(* IEC 61131-3 sources: AI4Industrial_Automation-FIRE2026/RUN-fih-02/taskA-outputs, 30 files *)

(* ---- task_01.st ---- *)
PROGRAM TankFillControl
VAR_INPUT
    Start_Button : BOOL;
    Stop_Button : BOOL;
    Low_Level_Sensor : BOOL;
    High_Level_Sensor : BOOL;
END_VAR
VAR_OUTPUT
    Fill_Pump : BOOL;
END_VAR
Fill_Pump := Start_Button AND NOT Low_Level_Sensor AND NOT High_Level_Sensor;
END_PROGRAM

(* ---- task_02.st ---- *)
PROGRAM traffic_light_cycle
VAR_OUTPUT
    Red_Light : BOOL;
    Yellow_Light : BOOL;
    Green_Light : BOOL;
END_VAR
VAR
    TP_Red : TP;
    TP_Yellow : TP;
    TP_Green : TP;
END_VAR
TP_Red(IN := TRUE, PT := T#5s);
TP_Yellow(IN := TRUE, PT := T#2s);
TP_Green(IN := TRUE, PT := T#5s);
Red_Light := TP_Red.Q;
Yellow_Light := TP_Yellow.Q;
Green_Light := TP_Green.Q;
END_PROGRAM

(* ---- task_03.st ---- *)
PROGRAM program0
VAR_INPUT
    Start_Button : BOOL;
    Stop_Button : BOOL;
    Overload_Trip : BOOL;
    Reset_Button : BOOL;
END_VAR
VAR_OUTPUT
    Motor_Run : BOOL;
    Fault_Lamp : BOOL;
END_VAR
VAR
    TON0 : TON;
END_VAR
TON0(IN := NOT Fault_Lamp AND (Start_Button OR Stop_Button), PT := T#5s);
Motor_Run := TON0.Q;
Fault_Lamp := Overload_Trip AND NOT TON0.Q;
END_PROGRAM

(* ---- task_04.st ---- *)
PROGRAM fill_cycle
VAR_INPUT
    Start_Button : BOOL;
    Stop_Button : BOOL;
    Bottle_Present : BOOL;
    Level_Sensor : BOOL;
END_VAR
VAR_OUTPUT
    Fill_Valve : BOOL;
END_VAR
VAR
    Cycle_Start : BOOL;
END_VAR
Cycle_Start := (Bottle_Present OR Level_Sensor) AND NOT Fill_Valve;
IF Cycle_Start THEN
    Fill_Valve := TRUE;
    Bottle_Count := Bottle_Count + 1;
END_IF;
Cycle_Start := FALSE;
END_PROGRAM

(* ---- task_05.st ---- *)
PROGRAM augerMotorControl
VAR_INPUT
    High_Level_Sensor : BOOL;
    Low_Level_Sensor : BOOL;
    Auto_Mode : BOOL;
END_VAR
VAR_OUTPUT
    Auger_Motor : BOOL;
    High_Alarm : BOOL;
END_VAR
VAR
    TON_high_alarm : TON;
END_VAR
TON_high_alarm(IN := High_Level_Sensor AND NOT High_Alarm, PT := T#10s);
High_Alarm := TON_high_alarm.Q;
Auger_Motor := Low_Level_Sensor AND Auto_Mode;
END_PROGRAM

(* ---- task_06.st ---- *)
PROGRAM program0
VAR_INPUT
    Start_Button : BOOL;
    Stop_Button : BOOL;
    E_Stop : BOOL;
    Reset_Button : BOOL;
END_VAR
VAR_OUTPUT
    Motor_Run : BOOL;
END_VAR
Motor_Run := NOT E_Stop AND NOT Stop_Button;
END_PROGRAM

(* ---- task_07.st ---- *)
PROGRAM conveyorControl
VAR_INPUT
    Start_Button : BOOL;
    Stop_Button : BOOL;
    Speed_Select : BOOL;
END_VAR
VAR_OUTPUT
    Running_Lamp : BOOL;
END_VAR
VAR
    conveyorStopped : BOOL;
    speedMode : BOOL;
END_VAR
conveyorStopped := Start_Button OR Stop_Button;
IF conveyorStopped THEN
    speedMode := FALSE;
    Conveyor_Speed := 0;
    Running_Lamp := FALSE;
ELSIF Speed_Select = TRUE THEN
    speedMode := TRUE;
    Conveyor_Speed := High_Speed_Set;
    Running_Lamp := TRUE;
END_IF;
IF speedMode THEN
    Conveyor_Speed := Low_Speed_Set;
END_IF;
END_PROGRAM

(* ---- task_08.st ---- *)
PROGRAM MultiValveCycle
VAR_INPUT
    Start_Button : BOOL;
    Reset_Button : BOOL;
    Level_A_Full : BOOL;
    Level_B_Full : BOOL;
END_VAR
VAR_OUTPUT
    Ingredient_A_Valve : BOOL;
    Ingredient_B_Valve : BOOL;
    Mixer_Motor : BOOL;
    Batch_Complete : BOOL;
END_VAR
VAR
    TON_Mixing : TON;
    scaled_level_a : REAL;
    scaled_level_b : REAL;
END_VAR
scaled_level_a := Level_A_Full / 50.0;
scaled_level_b := Level_B_Full / 50.0;
Ingredient_A_Valve := scaled_level_a >= 49.0 AND NOT Batch_Complete;
Ingredient_B_Valve := scaled_level_b >= 49.0 AND NOT Batch_Complete;
TON_Mixing(IN := Start_Button AND NOT Batch_Complete OR Reset_Button, PT := T#30s);
Mixer_Motor := TON_Mixing.Q;
Batch_Complete := Mixer_Motor OR Reset_Button;
END_PROGRAM

(* ---- task_09.st ---- *)
PROGRAM program0
VAR_INPUT
    Open_Button : BOOL;
    Close_Button : BOOL;
    Open_Limit : BOOL;
    Closed_Limit : BOOL;
    Obstacle_Sensor : BOOL;
END_VAR
VAR_OUTPUT
    Door_Motor_Open : BOOL;
    Door_Motor_Close : BOOL;
END_VAR
Door_Motor_Open := NOT Obstacle_Sensor AND Open_Button;
Door_Motor_Close := Close_Button AND NOT Open_Limit;
END_PROGRAM

(* ---- task_10.st ---- *)
PROGRAM Auto_CycleControl
VAR_INPUT
    Car_Present : BOOL;
    Start_Button : BOOL;
END_VAR
VAR_OUTPUT
    Wash_Pump : BOOL;
    Rinse_Valve : BOOL;
    Dryer_Fan : BOOL;
    Cycle_Complete : BOOL;
END_VAR
VAR
    TON_Wash : TON;
    TON_Rinse : TON;
    TON_Dry : TON;
END_VAR
TON_Wash(IN := Car_Present AND Start_Button, PT := T#20s);
TON_Rinse(IN := Car_Present AND Start_Button, PT := T#15s);
TON_Dry(IN := Car_Present AND Start_Button, PT := T#10s);
Wash_Pump := TON_Wash.Q;
Rinse_Valve := TON_Rinse.Q;
Dryer_Fan := TON_Dry.Q;
Cycle_Complete := TON_Dry.Q;
END_PROGRAM

(* ---- task_11.st ---- *)
PROGRAM program0
VAR_INPUT
    Box_Sensor : BOOL;
END_VAR
VAR_OUTPUT
    Pusher_Cylinder : BOOL;
    Box_Count_Display : BOOL;
END_VAR
VAR
    CTU0 : CTU;
    R_TRIG0 : R_TRIG;
    TP0 : TP;
END_VAR
R_TRIG0(CLK := Box_Sensor);
CTU0(CU := R_TRIG0.Q, R := FALSE, PV := 5);
TP0(IN := CTU0.Q, PT := T#1s);
Pusher_Cylinder := TP0.Q;
Box_Count_Display := CTU0.CV;
END_PROGRAM

(* ---- task_12.st ---- *)
PROGRAM weight_check
VAR_INPUT
    Weight_Input : INT;
    Target_Weight : INT;
    Photo_Eye : BOOL;
END_VAR
VAR_OUTPUT
    Reject_Pusher : BOOL;
END_VAR
VAR
    TON0 : TON;
END_VAR
TON0(IN := ABS(Weight_Input - Target_Weight) <= 500, PT := T#500MS);
Reject_Pusher := Photo_Eye AND NOT TON0.Q;
END_PROGRAM

(* ---- task_13.st ---- *)
PROGRAM HeatControl
VAR_INPUT
    Temp_Sensor : INT;
    Setpoint : INT;
END_VAR
VAR_OUTPUT
    Heater : BOOL;
END_VAR
VAR
    last_temp : INT;
    TON_heater_on : TON;
    TON_heater_off : TON;
END_VAR
TON_heater_on.et := Temp_Sensor - last_temp;
last_temp := Temp_Sensor;
TON_heater_on(IN := TON_heater_on.et <= 5, PT := T#1s);
TON_heater_off(IN := TON_heater_on.et >= 5, PT := T#1s);
IF TON_heater_on.Q THEN
    Heater := TRUE;
ELSIF TON_heater_off.Q THEN
    Heater := FALSE;
END_IF;
Heater := Heater AND (Temp_Sensor <= Setpoint + 5 OR Temp_Sensor >= Setpoint - 5);
END_PROGRAM

(* ---- task_14.st ---- *)
PROGRAM Temp_Controller
VAR_INPUT
    Temp_Sensor : INT;
END_VAR
VAR_OUTPUT
    Fan1 : BOOL;
    Fan2 : BOOL;
END_VAR
Fan1 := Temp_Sensor >= 300 AND Temp_Sensor <= 280;
Fan2 := Temp_Sensor >= 350 AND Temp_Sensor <= 330;
END_PROGRAM

(* ---- task_15.st ---- *)
PROGRAM compressorMotorControl
VAR_INPUT
    pressure_sensor : INT;
END_VAR
VAR_OUTPUT
    compressor_motor : BOOL;
END_VAR
compressor_motor := pressure_sensor >= 120 OR pressure_sensor <= 80;
END_PROGRAM

(* ---- task_16.st ---- *)
PROGRAM DamperControl
VAR_INPUT
    CO2_Sensor : INT;
END_VAR
VAR_OUTPUT
    Damper_Position : INT;
END_VAR
VAR
    TON_open : TON;
    TON_close : TON;
END_VAR
TON_open(IN := CO2_Sensor >= 1000, PT := T#10s);
TON_close(IN := CO2_Sensor <= 600, PT := T#10s);
IF TON_open.Q THEN
    Damper_Position := 100;
ELSIF TON_close.Q THEN
    Damper_Position := 0;
END_IF;
Damper_Position := Damper_Position + (CO2_Sensor - 600) / 400 * 2;
END_PROGRAM

(* ---- task_17.st ---- *)
PROGRAM IrrigationValveControl
VAR_INPUT
    soil_moisture : INT;
    manual_start : BOOL;
END_VAR
VAR_OUTPUT
    irrigation_valve : BOOL;
END_VAR
VAR
    TON_open : TON;
END_VAR
TON_open(IN := soil_moisture < 30 OR manual_start, PT := T#10s);
irrigation_valve := TON_open.Q AND NOT TON_open.et;
END_PROGRAM

(* ---- task_18.st ---- *)
PROGRAM PartDetect
VAR_INPUT
    Part_Detect : BOOL;
    Part_Good : BOOL;
END_VAR
VAR_OUTPUT
    Reject_Cylinder : BOOL;
END_VAR
VAR
    TON0 : TON;
END_VAR
TON0(IN := Part_Detect, PT := T#2s);
Reject_Cylinder := TON0.Q;
END_PROGRAM

(* ---- task_19.st ---- *)
PROGRAM ElevatorControl
VAR_INPUT
    call_floor1 : BOOL;
    call_floor2 : BOOL;
    at_floor1 : BOOL;
    at_floor2 : BOOL;
END_VAR
VAR_OUTPUT
    motor_up : BOOL;
    motor_down : BOOL;
END_VAR
VAR
    floor_sensor1 : BOOL;
    floor_sensor2 : BOOL;
    current_floor : INT;
    last_motor_up : BOOL;
    last_motor_down : BOOL;
END_VAR
floor_sensor1 := at_floor1;
floor_sensor2 := at_floor2;
IF call_floor1 AND NOT at_floor1 THEN
    current_floor := 1;
    motor_up := TRUE;
    motor_down := FALSE;
    last_motor_up := TRUE;
    last_motor_down := FALSE;
ELSIF call_floor2 AND NOT at_floor2 THEN
    current_floor := 2;
    motor_up := FALSE;
    motor_down := TRUE;
    last_motor_up := FALSE;
    last_motor_down := TRUE;
END_IF;
IF current_floor = 1 THEN
    motor_up := FALSE;
    motor_down := TRUE;
ELSIF current_floor = 2 THEN
    motor_up := FALSE;
    motor_down := FALSE;
END_IF;
IF last_motor_up AND NOT motor_up THEN
    motor_up := TRUE;
ELSIF last_motor_down AND NOT motor_down THEN
    motor_down := TRUE;
END_IF;
END_PROGRAM

(* ---- task_20.st ---- *)
PROGRAM CycleControl
VAR_INPUT
    Start_Cycle : BOOL;
    Part_Present : BOOL;
END_VAR
VAR_OUTPUT
    Gripper_Extended : BOOL;
    Gripper_Close : BOOL;
    Cylinder_Extend : BOOL;
END_VAR
VAR
    cycle_start : BOOL;
    grip_close : BOOL;
    wait_ms : TON;
END_VAR
cycle_start := Start_Cycle AND Part_Present;
grip_close := cycle_start AND Gripper_Extended;
IF grip_close THEN
    Gripper_Close := TRUE;
    wait_ms(IN := T#500ms);
    Gripper_Close := FALSE;
    Gripper_Extended := FALSE;
    Cylinder_Extend := FALSE;
END_IF;
Gripper_Extended := cycle_start OR grip_close;
Cylinder_Extend := cycle_start;
wait_ms(IN := wait_ms.Q);
END_PROGRAM

(* ---- task_21.st ---- *)
PROGRAM conveyor_control
VAR_INPUT
    Stop_Button : BOOL;
    Light_Curtain_Clear : BOOL;
END_VAR
VAR_OUTPUT
    Conveyor_Run : BOOL;
END_VAR
Conveyor_Run := Light_Curtain_Clear AND NOT Stop_Button;
END_PROGRAM

(* ---- task_22.st ---- *)
PROGRAM program0
VAR_INPUT
    Start_Button : BOOL;
    Stop_Button : BOOL;
    Entry_Photo_Eye : BOOL;
    Exit_Photo_Eye : BOOL;
END_VAR
VAR_OUTPUT
    Conveyor_Run : BOOL;
    Jam_Alarm : BOOL;
END_VAR
VAR
    TON_Jam : TON;
END_VAR
TON_Jam(IN := NOT Jam_Alarm AND Entry_Photo_Eye AND (NOT Stop_Button AND Exit_Photo_Eye), PT := T#8s);
Conveyor_Run := NOT TON_Jam.Q;
Jam_Alarm := Jam_Alarm OR TON_Jam.Q;
END_PROGRAM

(* ---- task_23.st ---- *)
PROGRAM DosingControl
VAR_INPUT
    Start_Button : BOOL;
    Stop_Button : BOOL;
    Flow_A_Pulse : BOOL;
END_VAR
VAR_OUTPUT
    Valve_A : BOOL;
    Valve_B : BOOL;
END_VAR
VAR
    CTU0 : CTU;
    R_TRIG0 : R_TRIG;
    TP0 : TP;
    TON0 : TON;
END_VAR
R_TRIG0(CLK := Flow_A_Pulse);
CTU0(CU := R_TRIG0.Q, R := FALSE, PV := 500);
TP0(IN := Start_Button AND NOT Stop_Button, PT := T#1s);
Valve_A := TP0.Q;
TON0(IN := TP0.Q, PT := T#1s);
Valve_B := TP0.Q AND (CTU0.CV * 1 + 1) MOD 4 = 1;
Valve_B := Valve_B OR TON0.Q;
END_PROGRAM

(* ---- task_24.st ---- *)
PROGRAM LightChaseControl
VAR_INPUT
    Start_Button : BOOL;
    Stop_Button : BOOL;
END_VAR
VAR_OUTPUT
    Lamp1 : BOOL;
    Lamp2 : BOOL;
    Lamp3 : BOOL;
    Lamp4 : BOOL;
END_VAR
VAR
    CTU0 : CTU;
    R_TRIG0 : R_TRIG;
    TP0 : TP;
END_VAR
R_TRIG0(CLK := Start_Button);
CTU0(CU := R_TRIG0.Q, R := Stop_Button, PV := 4);
IF CTU0.Q THEN
    TP0(IN := TRUE, PT := T#500ms);
    Lamp1 := TP0.Q;
    Lamp2 := Lamp1;
    Lamp3 := Lamp2;
    Lamp4 := Lamp3;
END_IF;
Lamp1 := NOT Lamp1;
Lamp2 := NOT Lamp2;
Lamp3 := NOT Lamp3;
Lamp4 := NOT Lamp4;
END_PROGRAM

(* ---- task_25.st ---- *)
PROGRAM pHControl
VAR_INPUT
    pH_Sensor : INT;
END_VAR
VAR_OUTPUT
    Acid_Pump : BOOL;
    Base_Pump : BOOL;
END_VAR
VAR
    TON_acid : TON;
    TON_base : TON;
END_VAR
TON_acid(IN := pH_Sensor > 720, PT := T#5s);
TON_base(IN := pH_Sensor < 680, PT := T#5s);
Acid_Pump := TRUE;
Base_Pump := FALSE;
IF TON_acid.Q THEN
    Acid_Pump := TRUE;
    Base_Pump := FALSE;
ELSIF TON_base.Q THEN
    Acid_Pump := FALSE;
    Base_Pump := TRUE;
END_IF;
END_PROGRAM

(* ---- task_26.st ---- *)
PROGRAM program0
VAR_INPUT
    Start_Button : BOOL;
    Stop_Button : BOOL;
END_VAR
VAR_OUTPUT
    Conveyor_Run : BOOL;
END_VAR
Conveyor_Run := Start_Button AND NOT Stop_Button;
END_PROGRAM

(* ---- task_27.st ---- *)
PROGRAM program0
VAR_INPUT
    Start_Button : BOOL;
    Stop_Button : BOOL;
END_VAR
VAR_OUTPUT
    Conveyor_Run : BOOL;
    Start_Light : BOOL;
END_VAR
VAR
    RPM_Set : INT;
END_VAR
RPM_Set := CONveyor_Run;
Conveyor_Run := Start_Button AND (RPM_Set OR NOT Stop_Button);
Start_Light := Conveyor_Run;
END_PROGRAM

(* ---- task_28.st ---- *)
PROGRAM program0
VAR_INPUT
    Start_Button : BOOL;
    Stop_Button : BOOL;
    RPM_Set : INT;
END_VAR
VAR_OUTPUT
    Conveyor_Run : BOOL;
    Digital_Display : INT;
END_VAR
VAR
    TON_Conveyor : TON;
END_VAR
TON_Conveyor(IN := Start_Button AND NOT TON_Conveyor.Q, PT := T#2s);
RPM_RPM := RPM_Set;
Digital_Display := RPM_RPM;
Conveyor_Run := TON_Conveyor.Q;
END_PROGRAM

(* ---- task_29.st ---- *)
PROGRAM program0
VAR_INPUT
    start_button : BOOL;
    stop_button : BOOL;
    vision_sensor : INT;
END_VAR
VAR_OUTPUT
    conveyor_run : BOOL;
    digital_display : BOOL;
    start_light : BOOL;
    box_counter : INT;
END_VAR
VAR
    RPM_Set : INT;
    TON0 : TON;
END_VAR
RPM_Set := RPM_Set + 1;
TON0(IN := (start_button OR start_light) AND NOT TON0.Q, PT := T#5s);
IF TON0.Q THEN
    conveyor_run := TRUE;
    digital_display := TRUE;
    start_light := FALSE;
END_IF;
box_counter := vision_sensor;
RPM_Set := box_counter / 10;
start_light := FALSE;
END_PROGRAM

(* ---- task_30.st ---- *)
PROGRAM conveyor_control_program
VAR_INPUT
    start_button : BOOL;
    stop_button : BOOL;
    vision_sensor_blue : INT;
    vision_sensor_green : INT;
    vision_sensor_gray : INT;
END_VAR
VAR_OUTPUT
    conveyor_run : BOOL;
    digital_display : BOOL;
    start_light : BOOL;
    display_box_counter : INT;
    blue_box_counter : INT;
    grey_box_counter : INT;
    green_box_counter : INT;
END_VAR
conveyor_run := NOT stop_button AND start_button;
digital_display := conveyor_run;
start_light := start_button OR conveyor_run;
total_boxes := vision_sensor_blue + (vision_sensor_green + vision_sensor_gray);
display_box_counter := total_boxes;
blue_box_counter := vision_sensor_blue;
grey_box_counter := vision_sensor_gray;
green_box_counter := vision_sensor_green;
RPM_Set := total_boxes / 100.0;
END_PROGRAM
